// TIA Portal V17 export
// export: Created 2022-07-26T05:39:22.6772606Z, ExportSetting WithDefaults, WithReadOnly, DisplayName Totally Integrated Automation Portal, DisplayVersion V17, DisplayName TIA Portal Openness, DisplayVersion V17, DisplayName TIA Portal Version Control Interface, DisplayVersion V17, DisplayName SINAMICS Startdrive Advanced, DisplayVersion V17, DisplayName SINAMICS Startdrive G130, G150, S120, S150, SINAMICS MV, S210, DisplayVersion V17, DisplayName SINAMICS Startdrive G110M, G120, G120C, G120D, G120P, G115D, DisplayVersion V17, DisplayName STEP 7 Professional, DisplayVersion V17, DisplayName STEP 7 Safety, DisplayVersion V17, DisplayName WinCC Advanced, DisplayVersion V17, DisplayName SIMATIC Visualization Architect, DisplayVersion V17
Screen "Screen_2"  1366x768, Number=2
  ScreenLayer 
    FaceplateInstance "MTR_Icon_Raw_3" at 40,28 size 50x50  FaceplateTypeName=IO@$@MTR@$@MTR_Icon_Raw V 0.0.5
      on CallPop: Motor_Popup_Parameters(Index := 1, X_Coordinates := 200, Y_Coordinates := 300)
      MTR := MTR_0001
    FaceplateInstance "MTR_Icon_Raw_1" at 127,28 size 50x50  FaceplateTypeName=IO@$@MTR@$@MTR_Icon_Raw V 0.0.5
      on CallPop: Motor_Popup_Parameters(Index := 2, X_Coordinates := 200, Y_Coordinates := 300)
      MTR := MTR_0002
